// TIA Portal V16 export
// export: Created 2024-05-10T06:46:44.3888498Z, ExportSetting WithDefaults, DisplayName Totally Integrated Automation Portal, DisplayVersion V16, DisplayName TIA Portal Version Control Interface, DisplayVersion V16, DisplayName TIA Portal Openness, DisplayVersion V16, DisplayName STEP 7 Professional, DisplayVersion V16, DisplayName STEP 7 Safety, DisplayVersion V16, DisplayName WinCC Professional, DisplayVersion V16
DATA_BLOCK "Com_DB"   // DB1
{ S7_Optimized_Access := 'TRUE' }
VERSION : 0.1
// stored: AutoNumber false, DBAccessibleFromOPCUA true, IsOnlyStoredInLoadMemory false, IsRetainMemResEnabled false, IsWriteProtectedInAS false, MemoryReserve 0
   VAR
      K01 : Struct   // S01使用
         "M" : Bool;
      END_STRUCT;
      K02 : Struct
         ST1_InitCont : Bool;   // ST1初始化条件
         ST1_InitStart : Bool;   // ST1初始化启动
      END_STRUCT;
      K03 : Struct
         InitTon2S { S7_SetPoint := 'True'} : IEC_TIMER;   // 初始2S
         PlcRunTon2s { S7_SetPoint := 'True'} : IEC_TIMER;   // 运行2秒
         PlcRunTon3s { S7_SetPoint := 'True'} : IEC_TIMER;   // 运行3秒
         PlcRunTon4s { S7_SetPoint := 'True'} : IEC_TIMER;   // 运行4秒
         EN_托盘在席 : Bool;
         EN_托盘离席 : Bool;
         EN_前端LS_ON { S7_SetPoint := 'True'} : IEC_TIMER;
         EN_前端LS_OFF { S7_SetPoint := 'True'} : IEC_TIMER;
         EN_后端LS_ON { S7_SetPoint := 'True'} : IEC_TIMER;
         EN_后端LS_OFF { S7_SetPoint := 'True'} : IEC_TIMER;
         EX_托盘在席 : Bool;
         EX_托盘离席 : Bool;
         EX_前端LS_ON { S7_SetPoint := 'True'} : IEC_TIMER;
         EX_前端LS_OFF { S7_SetPoint := 'True'} : IEC_TIMER;
         EX_后端LS_ON { S7_SetPoint := 'True'} : IEC_TIMER;
         EX_后端LS_OFF { S7_SetPoint := 'True'} : IEC_TIMER;
         ST01上托盘在席 : Bool;
         ST01上托盘离席 : Bool;
         ST01上前端LS_ON { S7_SetPoint := 'True'} : IEC_TIMER;
         ST01上前端LS_OFF { S7_SetPoint := 'True'} : IEC_TIMER;
         ST01上后端LS_ON { S7_SetPoint := 'True'} : IEC_TIMER;
         ST01上后端LS_OFF { S7_SetPoint := 'True'} : IEC_TIMER;
         ST01下托盘在席 : Bool;
         ST01下托盘离席 : Bool;
         ST01下前端LS_ON { S7_SetPoint := 'True'} : IEC_TIMER;
         ST01下前端LS_OFF { S7_SetPoint := 'True'} : IEC_TIMER;
         ST01下后端LS_ON { S7_SetPoint := 'True'} : IEC_TIMER;
         ST01下后端LS_OFF { S7_SetPoint := 'True'} : IEC_TIMER;
         ST02上托盘在席 : Bool;
         ST02上托盘离席 : Bool;
         ST02上前端LS_ON { S7_SetPoint := 'True'} : IEC_TIMER;
         ST02上前端LS_OFF { S7_SetPoint := 'True'} : IEC_TIMER;
         ST02上后端LS_ON { S7_SetPoint := 'True'} : IEC_TIMER;
         ST02上后端LS_OFF { S7_SetPoint := 'True'} : IEC_TIMER;
         ST02下托盘在席 : Bool;
         ST02下托盘离席 : Bool;
         ST02下前端LS_ON { S7_SetPoint := 'True'} : IEC_TIMER;
         ST02下前端LS_OFF { S7_SetPoint := 'True'} : IEC_TIMER;
         ST02下后端LS_ON { S7_SetPoint := 'True'} : IEC_TIMER;
         ST02下后端LS_OFF { S7_SetPoint := 'True'} : IEC_TIMER;
         ST03上托盘在席 : Bool;
         ST03上托盘离席 : Bool;
         ST03上前端LS_ON { S7_SetPoint := 'True'} : IEC_TIMER;
         ST03上前端LS_OFF { S7_SetPoint := 'True'} : IEC_TIMER;
         ST03上后端LS_ON { S7_SetPoint := 'True'} : IEC_TIMER;
         ST03上后端LS_OFF { S7_SetPoint := 'True'} : IEC_TIMER;
         ST03下托盘在席 : Bool;
         ST03下托盘离席 : Bool;
         ST03下前端LS_ON { S7_SetPoint := 'True'} : IEC_TIMER;
         ST03下前端LS_OFF { S7_SetPoint := 'True'} : IEC_TIMER;
         ST03下后端LS_ON { S7_SetPoint := 'True'} : IEC_TIMER;
         ST03下后端LS_OFF { S7_SetPoint := 'True'} : IEC_TIMER;
         ST04上托盘在席 : Bool;
         ST04上托盘离席 : Bool;
         ST04上前端LS_ON { S7_SetPoint := 'True'} : IEC_TIMER;
         ST04上前端LS_OFF { S7_SetPoint := 'True'} : IEC_TIMER;
         ST04上后端LS_ON { S7_SetPoint := 'True'} : IEC_TIMER;
         ST04上后端LS_OFF { S7_SetPoint := 'True'} : IEC_TIMER;
         ST05上托盘在席 : Bool;
         ST05上托盘离席 : Bool;
         ST05上前端LS_ON { S7_SetPoint := 'True'} : IEC_TIMER;
         ST05上前端LS_OFF { S7_SetPoint := 'True'} : IEC_TIMER;
         ST05上后端LS_ON { S7_SetPoint := 'True'} : IEC_TIMER;
         ST05上后端LS_OFF { S7_SetPoint := 'True'} : IEC_TIMER;
         ST06上托盘在席 : Bool;
         ST06上托盘离席 : Bool;
         ST06上前端LS_ON { S7_SetPoint := 'True'} : IEC_TIMER;
         ST06上前端LS_OFF { S7_SetPoint := 'True'} : IEC_TIMER;
         ST06上后端LS_ON { S7_SetPoint := 'True'} : IEC_TIMER;
         ST06上后端LS_OFF { S7_SetPoint := 'True'} : IEC_TIMER;
         ST07上托盘在席 : Bool;
         ST07上托盘离席 : Bool;
         ST07上前端LS_ON { S7_SetPoint := 'True'} : IEC_TIMER;
         ST07上前端LS_OFF { S7_SetPoint := 'True'} : IEC_TIMER;
         ST07上后端LS_ON { S7_SetPoint := 'True'} : IEC_TIMER;
         ST07上后端LS_OFF { S7_SetPoint := 'True'} : IEC_TIMER;
         ST08上托盘在席 : Bool;
         ST08上托盘离席 : Bool;
         ST08上前端LS_ON { S7_SetPoint := 'True'} : IEC_TIMER;
         ST08上前端LS_OFF { S7_SetPoint := 'True'} : IEC_TIMER;
         ST08上后端LS_ON { S7_SetPoint := 'True'} : IEC_TIMER;
         ST08上后端LS_OFF { S7_SetPoint := 'True'} : IEC_TIMER;
         ST09上托盘在席 : Bool;
         ST09上托盘离席 : Bool;
         ST09上前端LS_ON { S7_SetPoint := 'True'} : IEC_TIMER;
         ST09上前端LS_OFF { S7_SetPoint := 'True'} : IEC_TIMER;
         ST09上后端LS_ON { S7_SetPoint := 'True'} : IEC_TIMER;
         ST09上后端LS_OFF { S7_SetPoint := 'True'} : IEC_TIMER;
         ST10上托盘在席 : Bool;
         ST10上托盘离席 : Bool;
         ST10上前端LS_ON { S7_SetPoint := 'True'} : IEC_TIMER;
         ST10上前端LS_OFF { S7_SetPoint := 'True'} : IEC_TIMER;
         ST10上后端LS_ON { S7_SetPoint := 'True'} : IEC_TIMER;
         ST10上后端LS_OFF { S7_SetPoint := 'True'} : IEC_TIMER;
         ST11上托盘在席 : Bool;
         ST11上托盘离席 : Bool;
         ST11上前端LS_ON { S7_SetPoint := 'True'} : IEC_TIMER;
         ST11上前端LS_OFF { S7_SetPoint := 'True'} : IEC_TIMER;
         ST11上后端LS_ON { S7_SetPoint := 'True'} : IEC_TIMER;
         ST11上后端LS_OFF { S7_SetPoint := 'True'} : IEC_TIMER;
         ST12上托盘在席 : Bool;
         ST12上托盘离席 : Bool;
         ST12上前端LS_ON { S7_SetPoint := 'True'} : IEC_TIMER;
         ST12上前端LS_OFF { S7_SetPoint := 'True'} : IEC_TIMER;
         ST12上后端LS_ON { S7_SetPoint := 'True'} : IEC_TIMER;
         ST12上后端LS_OFF { S7_SetPoint := 'True'} : IEC_TIMER;
         ST01按压延迟 { S7_SetPoint := 'True'} : IEC_TIMER;
         ST02按压延迟 { S7_SetPoint := 'True'} : IEC_TIMER;
         ST03按压延迟 { S7_SetPoint := 'True'} : IEC_TIMER;
         ST04按压延迟 { S7_SetPoint := 'True'} : IEC_TIMER;
         ST05按压延迟 { S7_SetPoint := 'True'} : IEC_TIMER;
         ST06按压延迟 { S7_SetPoint := 'True'} : IEC_TIMER;
         ST07按压延迟 { S7_SetPoint := 'True'} : IEC_TIMER;
         ST08按压延迟 { S7_SetPoint := 'True'} : IEC_TIMER;
         ST09按压延迟 { S7_SetPoint := 'True'} : IEC_TIMER;
         ST10按压延迟 { S7_SetPoint := 'True'} : IEC_TIMER;
         ST11按压延迟 { S7_SetPoint := 'True'} : IEC_TIMER;
         ST12按压延迟 { S7_SetPoint := 'True'} : IEC_TIMER;
      END_STRUCT;
      K04 : Struct
         EMO : Array[1..16] of Bool;   // 急停报警
         SLC : Array[1..16] of Bool;   // 光栅报警
         DSW : Array[1..16] of Bool;   // 门SW报警
         OtherSafe : Array[1..16] of Bool;   // 其它安全报警
         AirALM : Array[1..16] of Bool;   // 气压报警
         AirALMTon : Array[1..16] of IEC_TIMER;   // 气压报警延迟
         DrumALM : Array[1..48] of Bool;   // 滚筒报警
         DrumTiOver : Array[1..48] of Bool;   // 滚筒超时
         DrumOverTon : Array[1..48] of IEC_TIMER;   // 滚筒超时延迟
         SensALM : Array[1..48] of Bool;   // 传感器故障
         SensTiOver : Array[1..48] of IEC_TIMER;   // 传感器故障延迟
         MoveALM : Array[1..48] of Bool;   // 动作异常
         MoveALMTiOver : Array[1..48] of IEC_TIMER;   // 动作异常延迟
         InvALM : Array[1..16] of Bool;   // 变频器故障
         InvNoRun : Array[1..16] of Bool;   // 变频器未运行故障
         InvNoRunTon : Array[1..16] of IEC_TIMER;   // 变频器未运行延迟
         InvTiOver : Array[1..16] of Bool;   // 变频器超时故障
         InvOverTon : Array[1..16] of IEC_TIMER;   // 变频器超时延迟
         InvOverload : Array[1..16] of Bool;   // 变频器过负载
         ValAdvTiOver : Array[1..48] of Bool;   // 阀出动作超时
         ValRetTiOver : Array[1..48] of Bool;   // 阀回动作超时
         ValSensALM : Array[1..48] of Bool;   // 阀到位传感器都ON故障
         ValSenCroALM : Array[1..48] of Bool;   // 阀到位传感器交叉ON故障
         AxisWarn : Array[1..16] of Bool;   // 轴警告
         AxisALM : Array[1..16] of Bool;   // 轴故障
         AxisNoReady : Array[1..16] of Bool;   // 轴未准备好
         AxisHomeALM : Array[1..16] of Bool;   // 轴未回零
         AxisNoRun : Array[1..16] of Bool;   // 轴未运行
         AxisNoRunTon : Array[1..16] of IEC_TIMER;   // 轴未运行超时
         AxisFLS : Array[1..16] of Bool;   // 轴正极限
         AxisRLS : Array[1..16] of Bool;   // 轴负极限
         RobotALM : Array[1..16] of Bool;   // 机器人故障
         CCDALM : Array[1..16] of Bool;   // 视觉故障
         CommALM : Array[1..16] of Bool;   // 通信故障
         AnalogUpALM : Array[1..16] of Bool;   // 模拟量上限故障
         AnalogLowALM : Array[1..16] of Bool;   // 模拟量下限故障
         OtherALM : Array[1..16] of Bool;   // 其它故障
      END_STRUCT;
      K05 : Struct
         ManTon { S7_SetPoint := 'True'} : IEC_TIMER;   // 手动延迟
         AutoTon { S7_SetPoint := 'True'} : IEC_TIMER;   // 自动延迟
      END_STRUCT;
      K06 : Struct
         AdvCond_Val { ExternalAccessible := 'False'; ExternalVisible := 'False'; ExternalWritable := 'False'} : Array[1..48] of Bool;   // 阀前进条件
         RetCond_Val { ExternalAccessible := 'False'; ExternalVisible := 'False'; ExternalWritable := 'False'} : Array[1..48] of Bool;   // 阀返回条件
         AdvCond_Drum { ExternalAccessible := 'False'; ExternalVisible := 'False'; ExternalWritable := 'False'} : Array[1..48] of Bool;   // 滚筒正转条件
         RetCond_Drum { ExternalAccessible := 'False'; ExternalVisible := 'False'; ExternalWritable := 'False'} : Array[1..48] of Bool;   // 滚筒反转条件
         AdvCond_Inv : Array[1..16] of Bool;   // 变频器正转条件
         RetCond_Inv : Array[1..16] of Bool;   // 变频器反转条件
      END_STRUCT;
      K07 : Struct
         Axis1Cont : Array[1..8] of Bool;   // 轴1动作条件
         Axis1Start : Bool;   // 轴1定位启动
         Axis1Pulse : Array[1..20] of Bool;   // 轴1脉冲
         Axis1Rate : Array[1..3] of Int;   // 轴1速率
         Axis1TON : Array[1..2] of IEC_TIMER;   // 轴1计时
         Axis2Cont : Array[1..8] of Bool;   // 轴2动作条件
         Axis2Start : Bool;   // 轴2定位启动
         Axis2Pulse : Array[1..20] of Bool;   // 轴2脉冲
         Axis2Rate : Array[1..3] of Int;   // 轴2速率
         Axis2TON : Array[1..2] of IEC_TIMER;   // 轴2计时
         Axis3Cont : Array[1..8] of Bool;   // 轴3动作条件
         Axis3Start : Bool;   // 轴3定位启动
         Axis3Pulse : Array[1..20] of Bool;   // 轴3脉冲
         Axis3Rate : Array[1..3] of Int;   // 轴3速率
         Axis3TON : Array[1..2] of IEC_TIMER;   // 轴3计时
         Axis4Cont : Array[1..8] of Bool;   // 轴4动作条件
         Axis4Start : Bool;   // 轴4定位启动
         Axis4Pulse : Array[1..20] of Bool;   // 轴4脉冲
         Axis4Rate : Array[1..3] of Int;   // 轴4速率
         Axis4TON : Array[1..2] of IEC_TIMER;   // 轴4计时
         Axis5Cont : Array[1..8] of Bool;   // 轴5动作条件
         Axis5Start : Bool;   // 轴5定位启动
         Axis5Pulse : Array[1..20] of Bool;   // 轴5脉冲
         Axis5Rate : Array[1..3] of Int;   // 轴5速率
         Axis5TON : Array[1..2] of IEC_TIMER;   // 轴5计时
         Axis6Cont : Array[1..8] of Bool;   // 轴6动作条件
         Axis6Start : Bool;   // 轴6定位启动
         Axis6Pulse : Array[1..20] of Bool;   // 轴6脉冲
         Axis6Rate : Array[1..3] of Int;   // 轴6速率
         Axis6TON : Array[1..2] of IEC_TIMER;   // 轴6计时
         Axis7Cont : Array[1..8] of Bool;   // 轴7动作条件
         Axis7Start : Bool;   // 轴7定位启动
         Axis7Pulse : Array[1..20] of Bool;   // 轴7脉冲
         Axis7Rate : Array[1..3] of Int;   // 轴7速率
         Axis7TON : Array[1..2] of IEC_TIMER;   // 轴7计时
         Axis8Cont : Array[1..8] of Bool;   // 轴8动作条件
         Axis8Start : Bool;   // 轴8定位启动
         Axis8Pulse : Array[1..20] of Bool;   // 轴8脉冲
         Axis8Rate : Array[1..3] of Int;   // 轴8速率
         Axis8TON : Array[1..2] of IEC_TIMER;   // 轴8计时
         Axis9Cont : Array[1..8] of Bool;   // 轴9动作条件
         Axis9Start : Bool;   // 轴9定位启动
         Axis9Pulse : Array[1..20] of Bool;   // 轴9脉冲
         Axis9Rate : Array[1..3] of Int;   // 轴9速率
         Axis9TON : Array[1..2] of IEC_TIMER;   // 轴9计时
         Axis10Cont : Array[1..8] of Bool;   // 轴10动作条件
         Axis10Start : Bool;   // 轴10定位启动
         Axis10Pulse : Array[1..20] of Bool;   // 轴10脉冲
         Axis10Rate : Array[1..3] of Int;   // 轴10速率
         Axis10TON : Array[1..2] of IEC_TIMER;   // 轴10计时
         Axis11Cont : Array[1..8] of Bool;   // 轴11动作条件
         Axis11Start : Bool;   // 轴11定位启动
         Axis11Pulse : Array[1..20] of Bool;   // 轴11脉冲
         Axis11Rate : Array[1..3] of Int;   // 轴11速率
         Axis11TON : Array[1..2] of IEC_TIMER;   // 轴11计时
         Axis12Cont : Array[1..8] of Bool;   // 轴12动作条件
         Axis12Start : Bool;   // 轴12定位启动
         Axis12Pulse : Array[1..20] of Bool;   // 轴12脉冲
         Axis12Rate : Array[1..3] of Int;   // 轴12速率
         Axis12TON : Array[1..2] of IEC_TIMER;   // 轴12计时
         Axis13Cont : Array[1..8] of Bool;   // 轴13动作条件
         Axis13Start : Bool;   // 轴13定位启动
         Axis13Pulse : Array[1..20] of Bool;   // 轴13脉冲
         Axis13Rate : Array[1..3] of Int;   // 轴13速率
         Axis13TON : Array[1..2] of IEC_TIMER;   // 轴13计时
         Axis14Cont : Array[1..8] of Bool;   // 轴14动作条件
         Axis14Start : Bool;   // 轴14定位启动
         Axis14Pulse : Array[1..20] of Bool;   // 轴4脉冲
         Axis14Rate : Array[1..3] of Int;   // 轴14速率
         Axis14TON : Array[1..2] of IEC_TIMER;   // 轴14计时
         Axis15Cont : Array[1..8] of Bool;   // 轴15动作条件
         Axis15Start : Bool;   // 轴15定位启动
         Axis15Pulse : Array[1..20] of Bool;   // 轴15脉冲
         Axis15Rate : Array[1..3] of Int;   // 轴15速率
         Axis15TON : Array[1..2] of IEC_TIMER;   // 轴15计时
         Axis16Cont : Array[1..8] of Bool;   // 轴16动作条件
         Axis16Start : Bool;   // 轴16定位启动
         Axis16Pulse : Array[1..20] of Bool;   // 轴16脉冲
         Axis16Rate : Array[1..3] of Int;   // 轴16速率
         Axis16TON : Array[1..2] of IEC_TIMER;   // 轴16计时
      END_STRUCT;
      K08 : Struct
         "M" : Bool;   // 位
      END_STRUCT;
      K10 : Struct
         "M" : Bool;   // 位
      END_STRUCT;
      K40 : Struct
         "M" : Bool;   // 位
      END_STRUCT;
   END_VAR
BEGIN
   // K04.ValAdvTiOver[1] : 阀1出动作超时
   // K04.ValAdvTiOver[2] : 阀2出动作超时
   // K04.ValAdvTiOver[3] : 阀3出动作超时
   // K04.ValAdvTiOver[4] : 阀4出动作超时
   // K04.ValAdvTiOver[5] : 阀5出动作超时
   // K04.ValAdvTiOver[6] : 阀6出动作超时
   // K04.ValAdvTiOver[7] : 阀7出动作超时
   // K04.ValAdvTiOver[8] : 阀8出动作超时
   // K04.ValRetTiOver[1] : 阀1回动作超时
   // K04.ValRetTiOver[2] : 阀2回动作超时
   // K04.ValRetTiOver[3] : 阀3回动作超时
   // K04.ValRetTiOver[4] : 阀4回动作超时
   // K04.ValRetTiOver[5] : 阀5回动作超时
   // K04.ValRetTiOver[6] : 阀6回动作超时
   // K04.ValRetTiOver[7] : 阀7回动作超时
   // K04.ValRetTiOver[8] : 阀8回动作超时
   // K06.AdvCond_Val[1] : 阀1前进条件
   // K06.AdvCond_Val[2] : 阀2前进条件
   // K06.AdvCond_Val[3] : 阀3前进条件
   // K06.AdvCond_Val[4] : 阀4前进条件
   // K06.AdvCond_Val[5] : 阀5前进条件
   // K06.AdvCond_Val[6] : 阀6前进条件
   // K06.AdvCond_Val[7] : 阀7前进条件
   // K06.AdvCond_Val[8] : 阀8前进条件
   // K06.AdvCond_Val[9] : 阀9前进条件
   // K06.AdvCond_Val[10] : 阀10前进条件
   // K06.AdvCond_Val[11] : 阀11前进条件
   // K06.AdvCond_Val[12] : 阀12前进条件
   // K06.AdvCond_Val[13] : 阀13前进条件
   // K06.AdvCond_Val[14] : 阀14前进条件
   // K06.AdvCond_Val[15] : 阀15前进条件
   // K06.AdvCond_Val[16] : 阀16前进条件
   // K06.AdvCond_Val[17] : 阀17前进条件
   // K06.AdvCond_Val[18] : 阀18前进条件
   // K06.AdvCond_Val[19] : 阀19前进条件
   // K06.AdvCond_Val[20] : 阀20前进条件
   // K06.AdvCond_Val[21] : 阀21前进条件
   // K06.AdvCond_Val[22] : 阀22前进条件
   // K06.AdvCond_Val[23] : 阀23前进条件
   // K06.AdvCond_Val[24] : 阀24前进条件
   // K06.AdvCond_Val[25] : 阀25前进条件
   // K06.AdvCond_Val[26] : 阀26前进条件
   // K06.AdvCond_Val[27] : 阀27前进条件
   // K06.AdvCond_Val[28] : 阀28前进条件
   // K06.AdvCond_Val[29] : 阀29前进条件
   // K06.AdvCond_Val[30] : 阀30前进条件
   // K06.AdvCond_Val[31] : 阀31前进条件
   // K06.AdvCond_Val[32] : 阀32前进条件
   // K06.AdvCond_Val[33] : 阀33前进条件
   // K06.AdvCond_Val[34] : 阀34前进条件
   // K06.AdvCond_Val[35] : 阀35前进条件
   // K06.AdvCond_Val[36] : 阀36前进条件
   // K06.AdvCond_Val[37] : 阀37前进条件
   // K06.AdvCond_Val[38] : 阀38前进条件
   // K06.AdvCond_Val[39] : 阀39前进条件
   // K06.AdvCond_Val[40] : 阀40前进条件
   // K06.AdvCond_Val[41] : 阀41前进条件
   // K06.AdvCond_Val[42] : 阀42前进条件
   // K06.AdvCond_Val[43] : 阀43前进条件
   // K06.AdvCond_Val[44] : 阀44前进条件
   // K06.AdvCond_Val[45] : 阀45前进条件
   // K06.AdvCond_Val[46] : 阀46前进条件
   // K06.AdvCond_Val[47] : 阀47前进条件
   // K06.AdvCond_Val[48] : 阀48前进条件
   // K06.RetCond_Val[1] : 阀1返回条件
   // K06.RetCond_Val[2] : 阀2返回条件
   // K06.RetCond_Val[3] : 阀3返回条件
   // K06.RetCond_Val[4] : 阀4返回条件
   // K06.RetCond_Val[5] : 阀5返回条件
   // K06.RetCond_Val[6] : 阀6返回条件
   // K06.RetCond_Val[7] : 阀7返回条件
   // K06.RetCond_Val[8] : 阀8返回条件
   // K06.RetCond_Val[9] : 阀9返回条件
   // K06.RetCond_Val[10] : 阀10返回条件
   // K06.RetCond_Val[11] : 阀11返回条件
   // K06.RetCond_Val[12] : 阀12返回条件
   // K06.RetCond_Val[13] : 阀13返回条件
   // K06.RetCond_Val[14] : 阀14返回条件
   // K06.RetCond_Val[15] : 阀15返回条件
   // K06.RetCond_Val[16] : 阀16返回条件
   // K06.RetCond_Val[17] : 阀17返回条件
   // K06.RetCond_Val[18] : 阀18返回条件
   // K06.RetCond_Val[19] : 阀19返回条件
   // K06.RetCond_Val[20] : 阀20返回条件
   // K06.RetCond_Val[21] : 阀21返回条件
   // K06.RetCond_Val[22] : 阀22返回条件
   // K06.RetCond_Val[23] : 阀23返回条件
   // K06.RetCond_Val[24] : 阀24返回条件
   // K06.RetCond_Val[25] : 阀25返回条件
   // K06.RetCond_Val[26] : 阀26返回条件
   // K06.RetCond_Val[27] : 阀27返回条件
   // K06.RetCond_Val[28] : 阀28返回条件
   // K06.RetCond_Val[29] : 阀29返回条件
   // K06.RetCond_Val[30] : 阀30返回条件
   // K06.RetCond_Val[31] : 阀31返回条件
   // K06.RetCond_Val[32] : 阀32返回条件
   // K06.RetCond_Val[33] : 阀33返回条件
   // K06.RetCond_Val[34] : 阀34返回条件
   // K06.RetCond_Val[35] : 阀35返回条件
   // K06.RetCond_Val[36] : 阀36返回条件
   // K06.RetCond_Val[37] : 阀37返回条件
   // K06.RetCond_Val[38] : 阀38返回条件
   // K06.RetCond_Val[39] : 阀39返回条件
   // K06.RetCond_Val[40] : 阀40返回条件
   // K06.RetCond_Val[41] : 阀41返回条件
   // K06.RetCond_Val[42] : 阀42返回条件
   // K06.RetCond_Val[43] : 阀43返回条件
   // K06.RetCond_Val[44] : 阀44返回条件
   // K06.RetCond_Val[45] : 阀45返回条件
   // K06.RetCond_Val[46] : 阀46返回条件
   // K06.RetCond_Val[47] : 阀47返回条件
   // K06.RetCond_Val[48] : 阀48返回条件
   // K07.Axis1Cont[1] : 共同条件
   // K07.Axis1Cont[2] : 回零条件
   // K07.Axis1Cont[3] : JOG正条件
   // K07.Axis1Cont[4] : JOG负条件
   // K07.Axis1Cont[5] : 定位正条件
   // K07.Axis1Cont[6] : 定位负条件
   // K07.Axis1Cont[7] : 预留
   // K07.Axis1Cont[8] : 预留
   // K07.Axis1Rate[1] : 轴1速率%
   // K07.Axis1Rate[2] : 轴1加速速率%
   // K07.Axis1Rate[3] : 轴1减速速率%
   // K07.Axis2Cont[1] : 共同条件
   // K07.Axis2Cont[2] : 回零条件
   // K07.Axis2Cont[3] : JOG正条件
   // K07.Axis2Cont[4] : JOG负条件
   // K07.Axis2Cont[5] : 定位正条件
   // K07.Axis2Cont[6] : 定位负条件
   // K07.Axis2Cont[7] : 预留
   // K07.Axis2Cont[8] : 预留
   // K07.Axis2Rate[1] : 轴1速率%
   // K07.Axis2Rate[2] : 轴1加速速率%
   // K07.Axis2Rate[3] : 轴1减速速率%
   // K07.Axis3Cont[1] : 共同条件
   // K07.Axis3Cont[2] : 回零条件
   // K07.Axis3Cont[3] : JOG正条件
   // K07.Axis3Cont[4] : JOG负条件
   // K07.Axis3Cont[5] : 定位正条件
   // K07.Axis3Cont[6] : 定位负条件
   // K07.Axis3Cont[7] : 预留
   // K07.Axis3Cont[8] : 预留
   // K07.Axis3Rate[1] : 轴1速率%
   // K07.Axis3Rate[2] : 轴1加速速率%
   // K07.Axis3Rate[3] : 轴1减速速率%
   // K07.Axis4Cont[1] : 共同条件
   // K07.Axis4Cont[2] : 回零条件
   // K07.Axis4Cont[3] : JOG正条件
   // K07.Axis4Cont[4] : JOG负条件
   // K07.Axis4Cont[5] : 定位正条件
   // K07.Axis4Cont[6] : 定位负条件
   // K07.Axis4Cont[7] : 预留
   // K07.Axis4Cont[8] : 预留
   // K07.Axis4Rate[1] : 轴1速率%
   // K07.Axis4Rate[2] : 轴1加速速率%
   // K07.Axis4Rate[3] : 轴1减速速率%
   // K07.Axis5Cont[1] : 共同条件
   // K07.Axis5Cont[2] : 回零条件
   // K07.Axis5Cont[3] : JOG正条件
   // K07.Axis5Cont[4] : JOG负条件
   // K07.Axis5Cont[5] : 定位正条件
   // K07.Axis5Cont[6] : 定位负条件
   // K07.Axis5Cont[7] : 预留
   // K07.Axis5Cont[8] : 预留
   // K07.Axis5Rate[1] : 轴1速率%
   // K07.Axis5Rate[2] : 轴1加速速率%
   // K07.Axis5Rate[3] : 轴1减速速率%
   // K07.Axis6Cont[1] : 共同条件
   // K07.Axis6Cont[2] : 回零条件
   // K07.Axis6Cont[3] : JOG正条件
   // K07.Axis6Cont[4] : JOG负条件
   // K07.Axis6Cont[5] : 定位正条件
   // K07.Axis6Cont[6] : 定位负条件
   // K07.Axis6Cont[7] : 预留
   // K07.Axis6Cont[8] : 预留
   // K07.Axis6Rate[1] : 轴1速率%
   // K07.Axis6Rate[2] : 轴1加速速率%
   // K07.Axis6Rate[3] : 轴1减速速率%
   // K07.Axis7Cont[1] : 共同条件
   // K07.Axis7Cont[2] : 回零条件
   // K07.Axis7Cont[3] : JOG正条件
   // K07.Axis7Cont[4] : JOG负条件
   // K07.Axis7Cont[5] : 定位正条件
   // K07.Axis7Cont[6] : 定位负条件
   // K07.Axis7Cont[7] : 预留
   // K07.Axis7Cont[8] : 预留
   // K07.Axis7Rate[1] : 轴1速率%
   // K07.Axis7Rate[2] : 轴1加速速率%
   // K07.Axis7Rate[3] : 轴1减速速率%
   // K07.Axis8Cont[1] : 共同条件
   // K07.Axis8Cont[2] : 回零条件
   // K07.Axis8Cont[3] : JOG正条件
   // K07.Axis8Cont[4] : JOG负条件
   // K07.Axis8Cont[5] : 定位正条件
   // K07.Axis8Cont[6] : 定位负条件
   // K07.Axis8Cont[7] : 预留
   // K07.Axis8Cont[8] : 预留
   // K07.Axis8Rate[1] : 轴1速率%
   // K07.Axis8Rate[2] : 轴1加速速率%
   // K07.Axis8Rate[3] : 轴1减速速率%
   // K07.Axis9Cont[1] : 共同条件
   // K07.Axis9Cont[2] : 回零条件
   // K07.Axis9Cont[3] : JOG正条件
   // K07.Axis9Cont[4] : JOG负条件
   // K07.Axis9Cont[5] : 定位正条件
   // K07.Axis9Cont[6] : 定位负条件
   // K07.Axis9Cont[7] : 预留
   // K07.Axis9Cont[8] : 预留
   // K07.Axis9Rate[1] : 轴1速率%
   // K07.Axis9Rate[2] : 轴1加速速率%
   // K07.Axis9Rate[3] : 轴1减速速率%
   // K07.Axis10Cont[1] : 共同条件
   // K07.Axis10Cont[2] : 回零条件
   // K07.Axis10Cont[3] : JOG正条件
   // K07.Axis10Cont[4] : JOG负条件
   // K07.Axis10Cont[5] : 定位正条件
   // K07.Axis10Cont[6] : 定位负条件
   // K07.Axis10Cont[7] : 预留
   // K07.Axis10Cont[8] : 预留
   // K07.Axis10Rate[1] : 轴1速率%
   // K07.Axis10Rate[2] : 轴1加速速率%
   // K07.Axis10Rate[3] : 轴1减速速率%
   // K07.Axis11Cont[1] : 共同条件
   // K07.Axis11Cont[2] : 回零条件
   // K07.Axis11Cont[3] : JOG正条件
   // K07.Axis11Cont[4] : JOG负条件
   // K07.Axis11Cont[5] : 定位正条件
   // K07.Axis11Cont[6] : 定位负条件
   // K07.Axis11Cont[7] : 预留
   // K07.Axis11Cont[8] : 预留
   // K07.Axis11Rate[1] : 轴1速率%
   // K07.Axis11Rate[2] : 轴1加速速率%
   // K07.Axis11Rate[3] : 轴1减速速率%
   // K07.Axis12Cont[1] : 共同条件
   // K07.Axis12Cont[2] : 回零条件
   // K07.Axis12Cont[3] : JOG正条件
   // K07.Axis12Cont[4] : JOG负条件
   // K07.Axis12Cont[5] : 定位正条件
   // K07.Axis12Cont[6] : 定位负条件
   // K07.Axis12Cont[7] : 预留
   // K07.Axis12Cont[8] : 预留
   // K07.Axis12Rate[1] : 轴1速率%
   // K07.Axis12Rate[2] : 轴1加速速率%
   // K07.Axis12Rate[3] : 轴1减速速率%
   // K07.Axis13Cont[1] : 共同条件
   // K07.Axis13Cont[2] : 回零条件
   // K07.Axis13Cont[3] : JOG正条件
   // K07.Axis13Cont[4] : JOG负条件
   // K07.Axis13Cont[5] : 定位正条件
   // K07.Axis13Cont[6] : 定位负条件
   // K07.Axis13Cont[7] : 预留
   // K07.Axis13Cont[8] : 预留
   // K07.Axis13Rate[1] : 轴1速率%
   // K07.Axis13Rate[2] : 轴1加速速率%
   // K07.Axis13Rate[3] : 轴1减速速率%
   // K07.Axis14Cont[1] : 共同条件
   // K07.Axis14Cont[2] : 回零条件
   // K07.Axis14Cont[3] : JOG正条件
   // K07.Axis14Cont[4] : JOG负条件
   // K07.Axis14Cont[5] : 定位正条件
   // K07.Axis14Cont[6] : 定位负条件
   // K07.Axis14Cont[7] : 预留
   // K07.Axis14Cont[8] : 预留
   // K07.Axis14Rate[1] : 轴1速率%
   // K07.Axis14Rate[2] : 轴1加速速率%
   // K07.Axis14Rate[3] : 轴1减速速率%
   // K07.Axis15Cont[1] : 共同条件
   // K07.Axis15Cont[2] : 回零条件
   // K07.Axis15Cont[3] : JOG正条件
   // K07.Axis15Cont[4] : JOG负条件
   // K07.Axis15Cont[5] : 定位正条件
   // K07.Axis15Cont[6] : 定位负条件
   // K07.Axis15Cont[7] : 预留
   // K07.Axis15Cont[8] : 预留
   // K07.Axis15Rate[1] : 轴1速率%
   // K07.Axis15Rate[2] : 轴1加速速率%
   // K07.Axis15Rate[3] : 轴1减速速率%
   // K07.Axis16Cont[1] : 共同条件
   // K07.Axis16Cont[2] : 回零条件
   // K07.Axis16Cont[3] : JOG正条件
   // K07.Axis16Cont[4] : JOG负条件
   // K07.Axis16Cont[5] : 定位正条件
   // K07.Axis16Cont[6] : 定位负条件
   // K07.Axis16Cont[7] : 预留
   // K07.Axis16Cont[8] : 预留
   // K07.Axis16Rate[1] : 轴1速率%
   // K07.Axis16Rate[2] : 轴1加速速率%
   // K07.Axis16Rate[3] : 轴1减速速率%
END_DATA_BLOCK
